(* CoDeSys 2.3 export: CHECKBOUNDS.EXP *)

(* POU CheckBounds, ST *)
FUNCTION CheckBounds : DINT
VAR_INPUT
	index, lower, upper: DINT;
END_VAR
VAR
END_VAR
(* @TEXT_IMPLEMENTATION := 'ST' *)
IF index < lower THEN
	CheckBounds := lower;
ELSIF index > upper THEN
	CheckBounds := upper;
ELSE CheckBounds := index;
END_IF
END_FUNCTION
